(* LS Electric XG5000 project: Sample *)
(* PLC NewPLC *)

PROGRAM DsLogic (* task: 스캔 프로그램 *)
VAR
    a : BOOL;
    b : BOOL;
    c : BOOL;
    d : BOOL;
    myBoolean : BOOL; (* BOOL <- Boolean *)
    mySingle : REAL; (* REAL <- Single *)
    myDouble : LREAL; (* LREAL <- Double *)
    mySByte : BYTE; (* BYTE <- SByte *)
    myChar : BYTE; (* BYTE <- Char *)
    myByte : BYTE; (* BYTE <- Byte *)
    myInt16 : INT; (* INT <- Int16 *)
    myUInt16 : INT; (* INT <- UInt16 *)
    myInt32 : DINT; (* DINT <- Int32 *)
    myUInt32 : DINT; (* DINT <- UInt32 *)
    myInt64 : LINT; (* LINT <- Int64 *)
    myUInt64 : LINT; (* LINT <- UInt64 *)
    myString : STRING; (* STRING <- String *)
    OrBy2 : BOOL;
END_VAR

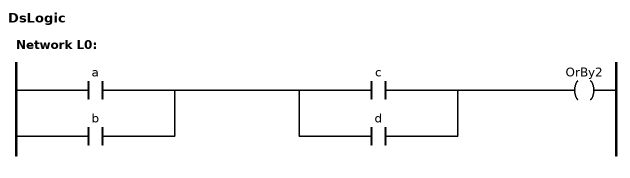
(* Rung L0 *)
OrBy2 := (a OR b) AND (c OR d);
END_PROGRAM